PROGRAM MobjectEventsUnitTests
VAR
	eventEmitter_TestSuite : EventEmitter_TestSuite;
	eventEmitterInterface_TestSuite : EventEmitterInterface_TestSuite;
	eventTargetInterface_TestSuite : EventTargetInterface_TestSuite;
	eventHandlerInterface_TestSuite : EventHandlerInterface_TestSuite;
END_VAR

END_PROGRAM

(* stored: Version 1.1.0.1, ProductVersion 3.1.4024.12
   POU MobjectEventsUnitTests: Id {f5065049-6869-034f-178d-2c0b223ac755}, SpecialFunc None *)
